Staubli VAL3: cmdAbortHoming.pgx

public program cmdAbortHoming(num x_nAxisNum)
begin
 //取消回零

end
